FUNCTION_BLOCK fb_level_ctrl

VAR_INPUT
END_VAR

VAR_OUTPUT
END_VAR

VAR
	stripper_level_dpi: fb_discrete_pi			:= (kc:=2E-4, ti:=200/60, Ts:=g_Ts_base, hi :=100, lo:=0, x0:=r_0[7]);
	separator_level_dpi: fb_discrete_pi			:= (kc:=-1E-3, ti:=200/60, Ts:=g_Ts_base, hi :=100, lo:=0, x0:=r_0[6]);
	reactor_level_dpi: fb_discrete_pi			:= (kc:=0.8, ti:=60/60, Ts:=g_Ts_base, hi :=100, lo:=0, x0:=SP17_0);
	reactor_pressure_dpi: fb_discrete_pi		:= (kc:=-1E-4, ti:=20/60, Ts:=g_Ts_base, hi :=100, lo:=0, x0:=r_0[5]);
	reactor_temp_dpi: fb_discrete_pi			:= (kc:=-8, ti:=7.5/60, Ts:=g_Ts_base, hi :=100, lo:=0, x0:=xmv_0[10]);		
END_VAR

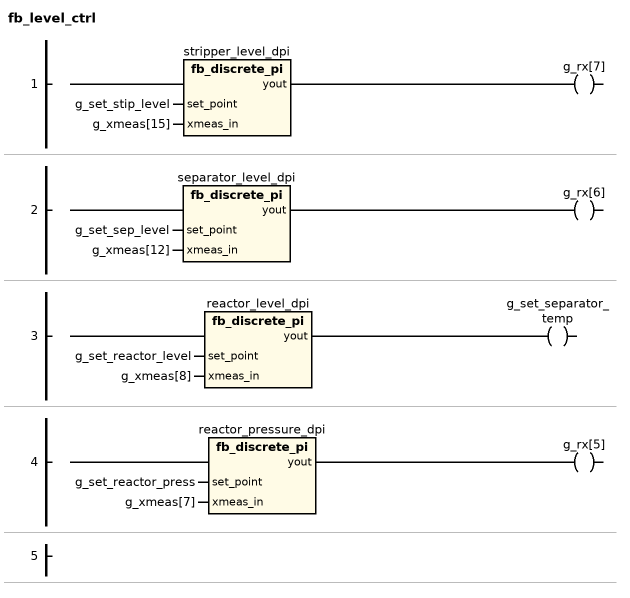
// NETWORK 1
//   g_xmeas[15]: storage variables for sub-controllers
stripper_level_dpi(set_point := g_set_stip_level, xmeas_in := g_xmeas[15]); // fb_discrete_pi
g_rx[7] := stripper_level_dpi.yout;

// NETWORK 2
//   g_xmeas[12]: storage variables for sub-controllers
separator_level_dpi(set_point := g_set_sep_level, xmeas_in := g_xmeas[12]); // fb_discrete_pi
g_rx[6] := separator_level_dpi.yout;

// NETWORK 3
//   g_xmeas[8]: storage variables for sub-controllers
reactor_level_dpi(set_point := g_set_reactor_level, xmeas_in := g_xmeas[8]); // fb_discrete_pi
g_set_separator_temp := reactor_level_dpi.yout;

// NETWORK 4
//   g_xmeas[7]: storage variables for sub-controllers
reactor_pressure_dpi(set_point := g_set_reactor_press, xmeas_in := g_xmeas[7]); // fb_discrete_pi
g_rx[5] := reactor_pressure_dpi.yout;

// NETWORK 5

END_FUNCTION_BLOCK

(* stored: Version 1.1.0.1, ProductVersion 3.1.0.26
   POU fb_level_ctrl: Id {ff448cf3-b526-4727-8e64-f2816dd51673} *)
